# B&R Automation Studio project MotionProyect (part 2)

#### basicCyclic.st - cyclic code
```iecst
(********************************************************************
 * COPYRIGHT -- Bernecker + Rainer
 ********************************************************************
 * PROGRAM: Basic
 * File: basicCyclic.st
 * Author: Bernecker + Rainer
 * Created: December 01, 2009
 ********************************************************************
 * Implementation of Program Basic
 ********************************************************************)
PROGRAM _CYCLIC

(***************************************************************
        Control Sequence
***************************************************************)
	Axis2Cmd;
	Axis2Param;
	Axis2CyclicReadAction;

(* status information is read before the step sequencer to attain a shorter reaction time *)
(************************ MC_READSTATUS *************************)
MC_ReadStatus_0.Enable := NOT(MC_ReadStatus_0.Error);
MC_ReadStatus_0.Axis := Axis1Obj;
MC_ReadStatus_0();
BasicControl.AxisState.Disabled             := MC_ReadStatus_0.Disabled;
BasicControl.AxisState.StandStill           := MC_ReadStatus_0.StandStill;
BasicControl.AxisState.Stopping             := MC_ReadStatus_0.Stopping;
BasicControl.AxisState.Homing               := MC_ReadStatus_0.Homing;
BasicControl.AxisState.DiscreteMotion       := MC_ReadStatus_0.DiscreteMotion;
BasicControl.AxisState.ContinuousMotion     := MC_ReadStatus_0.ContinuousMotion;
BasicControl.AxisState.SynchronizedMotion   := MC_ReadStatus_0.SynchronizedMotion;
BasicControl.AxisState.ErrorStop            := MC_ReadStatus_0.Errorstop;

(********************MC_BR_READDRIVESTATUS***********************)
MC_BR_ReadDriveStatus_0.Enable := NOT(MC_BR_ReadDriveStatus_0.Error);
MC_BR_ReadDriveStatus_0.Axis := Axis1Obj;
MC_BR_ReadDriveStatus_0.AdrDriveStatus := ADR(BasicControl.Status.DriveStatus);
MC_BR_ReadDriveStatus_0();

(******************** MC_READACTUALPOSITION *********************)
MC_ReadActualPosition_0.Enable := (NOT(MC_ReadActualPosition_0.Error));
MC_ReadActualPosition_0.Axis := Axis1Obj;
MC_ReadActualPosition_0();
IF(MC_ReadActualPosition_0.Valid = TRUE)THEN
    BasicControl.Status.ActPosition := MC_ReadActualPosition_0.Position;
END_IF

(******************** MC_READACTUALVELOCITY *********************)
MC_ReadActualVelocity_0.Enable := (NOT(MC_ReadActualVelocity_0.Error));
MC_ReadActualVelocity_0.Axis := Axis1Obj;
MC_ReadActualVelocity_0();
IF(MC_ReadActualVelocity_0.Valid = TRUE)THEN
    BasicControl.Status.ActVelocity := MC_ReadActualVelocity_0.Velocity;
END_IF

(************************ MC_READAXISERROR **********************)
MC_ReadAxisError_0.Enable := NOT(MC_ReadAxisError_0.Error);
MC_ReadAxisError_0.Axis := Axis1Obj;
MC_ReadAxisError_0.DataAddress := ADR(BasicControl.Status.ErrorText);
MC_ReadAxisError_0.DataLength := SIZEOF(BasicControl.Status.ErrorText);
MC_ReadAxisError_0.DataObjectName := 'acp10etxen';
MC_ReadAxisError_0();

(**************** CHECK FOR GENERAL AXIS ERROR ******************)
    IF ((MC_ReadAxisError_0.AxisErrorID <> 0) AND (MC_ReadAxisError_0.Valid = TRUE)) THEN
        AxisStep := STATE_ERROR_AXIS;
(***************** CHECK IF POWER SHOULD BE OFF *******************)
    ELSIF ((BasicControl.Command.Power = FALSE) AND (MC_ReadAxisError_0.Valid = TRUE)) THEN
        IF ((MC_ReadStatus_0.Errorstop = TRUE) AND (MC_ReadStatus_0.Valid = TRUE)) THEN
            AxisStep := STATE_ERROR_RESET;
        ELSE
            AxisStep := STATE_WAIT;
        END_IF
    END_IF

(* central monitoring OF stop command attains a shorter reaction TIME in CASE OF emergency stop *)
(******************CHECK FOR STOP COMMAND************************)
    IF (BasicControl.Command.Stop = TRUE) THEN
        IF ((AxisStep >= STATE_HOME) AND (AxisStep <= STATE_ERROR)) THEN
            (* reset all FB execute inputs we use *)
            MC_Home_0.Execute := 0;
            MC_Stop_0.Execute := 0;
            MC_MoveAbsolute_0.Execute := 0;
            MC_MoveAdditive_0.Execute := 0;
            MC_MoveVelocity_0.Execute := 0;
            MC_ReadAxisError_0.Acknowledge := 0;
            MC_Reset_0.Execute := 0;
            MC_Halt_0.Execute := 0;

            (* reset user commands *)
            BasicControl.Command.Halt := 0;
            BasicControl.Command.Home := 0;
            BasicControl.Command.MoveJogPos := 0;
            BasicControl.Command.MoveJogNeg := 0;
            BasicControl.Command.MoveVelocity := 0;
            BasicControl.Command.MoveAbsolute := 0;
            BasicControl.Command.MoveAdditive := 0;
            AxisStep := STATE_STOP;
        END_IF
    END_IF

CASE AxisStep OF

(******************** WAIT *************************)
    STATE_WAIT:  (* STATE: Wait *)
        IF (BasicControl.Command.Power = TRUE) THEN
            AxisStep := STATE_POWER_ON;
        ELSE
            MC_Power_0.Enable := FALSE;
        END_IF

        (* reset all FB execute inputs we use *)
        MC_Home_0.Execute := FALSE;
        MC_Stop_0.Execute := FALSE;
        MC_MoveAbsolute_0.Execute := FALSE;
        MC_MoveAdditive_0.Execute := FALSE;
        MC_MoveVelocity_0.Execute := FALSE;
        MC_Halt_0.Execute := FALSE;
        MC_ReadAxisError_0.Acknowledge := FALSE;
        MC_Reset_0.Execute := FALSE;

        (* reset user commands *)
        BasicControl.Command.Stop := FALSE;
        BasicControl.Command.Halt := FALSE;
        BasicControl.Command.Home := FALSE;
        BasicControl.Command.MoveJogPos := FALSE;
        BasicControl.Command.MoveJogNeg := FALSE;
        BasicControl.Command.MoveVelocity := FALSE;
        BasicControl.Command.MoveAbsolute := FALSE;
        BasicControl.Command.MoveAdditive := FALSE;

        BasicControl.Status.ErrorID := 0;

(******************** POWER ON **********************)
    STATE_POWER_ON:  (* STATE: Power on *)
        MC_Power_0.Enable := TRUE;
        IF (MC_Power_0.Status = TRUE) THEN
            AxisStep := STATE_READY;
        END_IF
        (* if a power error occured go to error state *)
        IF (MC_Power_0.Error = TRUE) THEN
            BasicControl.Status.ErrorID := MC_Power_0.ErrorID;
            AxisStep := STATE_ERROR;
        END_IF

(******************** READY **********************)
    STATE_READY:  (* STATE: Waiting for commands *)
        IF (BasicControl.Command.Home = TRUE)THEN
            BasicControl.Command.Home := FALSE;
            AxisStep := STATE_HOME;

        ELSIF (BasicControl.Command.Stop = TRUE) THEN
            AxisStep := STATE_STOP;

        ELSIF (BasicControl.Command.MoveJogPos = TRUE) THEN
            AxisStep := STATE_JOG_POSITIVE;

        ELSIF (BasicControl.Command.MoveJogNeg = TRUE) THEN
            AxisStep := STATE_JOG_NEGATIVE;

        ELSIF (BasicControl.Command.MoveAbsolute = TRUE) THEN
            BasicControl.Command.MoveAbsolute := FALSE;
            AxisStep := STATE_MOVE_ABSOLUTE;

        ELSIF (BasicControl.Command.MoveAdditive = TRUE) THEN
            BasicControl.Command.MoveAdditive := FALSE;
            AxisStep := STATE_MOVE_ADDITIVE;

        ELSIF (BasicControl.Command.MoveVelocity = TRUE) THEN
            BasicControl.Command.MoveVelocity := FALSE;
            AxisStep := STATE_MOVE_VELOCITY;

        ELSIF (BasicControl.Command.Halt = TRUE) THEN
            BasicControl.Command.Halt := FALSE;
            AxisStep := STATE_HALT;
        END_IF

(******************** HOME **********************)
    STATE_HOME:  (* STATE: start homing process *)
        MC_Home_0.Position := BasicControl.Parameter.HomePosition;
        MC_Home_0.HomingMode := BasicControl.Parameter.HomeMode;
        MC_Home_0.Execute := TRUE;
        IF (MC_Home_0.Done = TRUE) THEN
            MC_Home_0.Execute := FALSE;
            AxisStep := STATE_READY;
        END_IF
        (* if a homing error occured go to error state *)
        IF (MC_Home_0.Error = TRUE) THEN
            MC_Home_0.Execute := FALSE;
            BasicControl.Status.ErrorID := MC_Home_0.ErrorID;
            AxisStep := STATE_ERROR;
        END_IF

(***********************HALT_MOVEMENT***************************)
    STATE_HALT:   (* STATE: Halt movement *)
        MC_Halt_0.Deceleration := BasicControl.Parameter.Deceleration;
        MC_Halt_0.Execute := TRUE;
        IF (MC_Halt_0.Done = TRUE) THEN
            MC_Halt_0.Execute := FALSE;
            AxisStep := STATE_READY;
        END_IF
        (* check if error occured *)
        IF (MC_Halt_0.Error = TRUE) THEN
            BasicControl.Status.ErrorID := MC_Halt_0.ErrorID;
            MC_Halt_0.Execute := FALSE;
            AxisStep := STATE_ERROR;
        END_IF

(*********************** STOP MOVEMENT *************************)
    STATE_STOP:  (* STATE: Stop movement *)
        MC_Stop_0.Deceleration := BasicControl.Parameter.Deceleration;
        MC_Stop_0.Execute := TRUE;
        (* if axis is stopped go to ready state *)
        IF ((MC_Stop_0.Done = TRUE) AND (BasicControl.Command.Stop = FALSE)) THEN
            MC_Stop_0.Execute := FALSE;
            AxisStep := STATE_READY;
        END_IF
        (* check if error occured *)
        IF (MC_Stop_0.Error = TRUE) THEN
            BasicControl.Status.ErrorID := MC_Stop_0.ErrorID;
            MC_Stop_0.Execute := FALSE;
            AxisStep := STATE_ERROR;
        END_IF

(******************** START JOG MOVEMENT POSITVE **********************)
     STATE_JOG_POSITIVE:  (* STATE: Start jog movement in positive direction *)
        MC_MoveVelocity_0.Velocity      := BasicControl.Parameter.JogVelocity;
        MC_MoveVelocity_0.Acceleration  := BasicControl.Parameter.Acceleration;
        MC_MoveVelocity_0.Deceleration  := BasicControl.Parameter.Deceleration;
        MC_MoveVelocity_0.Direction     := mcPOSITIVE_DIR;
        MC_MoveVelocity_0.Execute := TRUE;
        IF (BasicControl.Command.MoveJogPos = FALSE) THEN
            MC_MoveVelocity_0.Execute := FALSE;
            AxisStep := STATE_HALT;
        END_IF
        (* check if error occured *)
        IF (MC_MoveVelocity_0.Error = TRUE) THEN
            BasicControl.Status.ErrorID := MC_MoveVelocity_0.ErrorID;
            MC_MoveVelocity_0.Execute := FALSE;
            AxisStep := STATE_ERROR;
        END_IF

(******************** START JOG MOVEMENT NEGATIVE **********************)
    STATE_JOG_NEGATIVE:  (* STATE: Start jog movement in negative direction *)
        MC_MoveVelocity_0.Velocity      := BasicControl.Parameter.JogVelocity;
        MC_MoveVelocity_0.Acceleration  := BasicControl.Parameter.Acceleration;
        MC_MoveVelocity_0.Deceleration  := BasicControl.Parameter.Deceleration;
        MC_MoveVelocity_0.Direction	    := mcNEGATIVE_DIR;
        MC_MoveVelocity_0.Execute := TRUE;
        IF (BasicControl.Command.MoveJogNeg = FALSE) THEN
            MC_MoveVelocity_0.Execute := FALSE;
            AxisStep := STATE_HALT;
        END_IF
        (* check if error occured *)
        IF (MC_MoveVelocity_0.Error = TRUE) THEN
            BasicControl.Status.ErrorID := MC_MoveVelocity_0.ErrorID;
            MC_MoveVelocity_0.Execute := FALSE;
            AxisStep := STATE_ERROR;
        END_IF

(******************** START ABSOLUTE MOVEMENT **********************)
     STATE_MOVE_ABSOLUTE:  (* STATE: Start absolute movement *)
        MC_MoveAbsolute_0.Position      := BasicControl.Parameter.Position;
        MC_MoveAbsolute_0.Velocity      := BasicControl.Parameter.Velocity;
        MC_MoveAbsolute_0.Acceleration  := BasicControl.Parameter.Acceleration;
        MC_MoveAbsolute_0.Deceleration  := BasicControl.Parameter.Deceleration;
        MC_MoveAbsolute_0.Direction     := BasicControl.Parameter.Direction;
        MC_MoveAbsolute_0.Execute := TRUE;
        (* check if commanded position is reached *)
        IF (BasicControl.Command.Halt) THEN
            BasicControl.Command.Halt := FALSE;
            MC_MoveAbsolute_0.Execute := FALSE;
            AxisStep := STATE_HALT;
        ELSIF (MC_MoveAbsolute_0.Done = TRUE) THEN
            MC_MoveAbsolute_0.Execute := FALSE;
            AxisStep := STATE_READY;
        END_IF
        (* check if error occured *)
        IF (MC_MoveAbsolute_0.Error = TRUE) THEN
            BasicControl.Status.ErrorID := MC_MoveAbsolute_0.ErrorID;
            MC_MoveAbsolute_0.Execute := FALSE;
            AxisStep := STATE_ERROR;
        END_IF

(******************** START ADDITIVE MOVEMENT **********************)
    STATE_MOVE_ADDITIVE:  (* STATE: Start additive movement *)
        MC_MoveAdditive_0.Distance      := BasicControl.Parameter.Distance;
        MC_MoveAdditive_0.Velocity      := BasicControl.Parameter.Velocity;
        MC_MoveAdditive_0.Acceleration  := BasicControl.Parameter.Acceleration;
        MC_MoveAdditive_0.Deceleration  := BasicControl.Parameter.Deceleration;
        MC_MoveAdditive_0.Execute := TRUE;
        (* check if commanded distance is reached *)
        IF (BasicControl.Command.Halt) THEN
            BasicControl.Command.Halt := FALSE;
            MC_MoveAdditive_0.Execute := FALSE;
            AxisStep := STATE_HALT;
        ELSIF (MC_MoveAdditive_0.Done = TRUE) THEN
            MC_MoveAdditive_0.Execute := FALSE;
            AxisStep := STATE_READY;
        END_IF
        (* check if error occured *)
        IF (MC_MoveAdditive_0.Error = TRUE) THEN
            BasicControl.Status.ErrorID := MC_MoveAdditive_0.ErrorID;
            MC_MoveAdditive_0.Execute := FALSE;
            AxisStep := STATE_ERROR;
        END_IF

(******************** START VELOCITY MOVEMENT **********************)
    STATE_MOVE_VELOCITY:  (* STATE: Start velocity movement *)
        MC_MoveVelocity_0.Velocity      := BasicControl.Parameter.Velocity;
        MC_MoveVelocity_0.Acceleration  := BasicControl.Parameter.Acceleration;
        MC_MoveVelocity_0.Deceleration  := BasicControl.Parameter.Deceleration;
        MC_MoveVelocity_0.Direction     := BasicControl.Parameter.Direction;
        MC_MoveVelocity_0.Execute := TRUE;
        (* check if commanded velocity is reached *)
        IF (BasicControl.Command.Halt) THEN
            BasicControl.Command.Halt := FALSE;
            MC_MoveVelocity_0.Execute := FALSE;
            AxisStep := STATE_HALT;
        ELSIF (MC_MoveVelocity_0.InVelocity = TRUE) THEN
            MC_MoveVelocity_0.Execute := FALSE;
            AxisStep := STATE_READY;
        END_IF
        (* check if error occured *)
        IF (MC_MoveVelocity_0.Error = TRUE) THEN
            BasicControl.Status.ErrorID := MC_MoveVelocity_0.ErrorID;
            MC_MoveVelocity_0.Execute := FALSE;
            AxisStep := STATE_ERROR;
        END_IF

(******************** FB-ERROR OCCURED *************************)
    STATE_ERROR:  (* STATE: Error *)
        (* check if FB indicates an axis error *)
        IF (MC_ReadAxisError_0.AxisErrorCount<>0) THEN
            AxisStep := STATE_ERROR_AXIS;
        ELSE
            IF (BasicControl.Command.ErrorAcknowledge = TRUE) THEN
                BasicControl.Command.ErrorAcknowledge := FALSE;
                BasicControl.Status.ErrorID := 0;
                (* reset axis if it is in axis state ErrorStop *)
                IF ((MC_ReadStatus_0.Errorstop = TRUE) AND (MC_ReadStatus_0.Valid = TRUE)) THEN
                    AxisStep := STATE_ERROR_RESET;
                ELSE
                    AxisStep := STATE_WAIT;
                END_IF
            END_IF
        END_IF

(******************** AXIS-ERROR OCCURED *************************)
    STATE_ERROR_AXIS:  (* STATE: Axis Error *)
        IF (MC_ReadAxisError_0.Valid = TRUE) THEN
            IF (MC_ReadAxisError_0.AxisErrorID <> 0) THEN
                BasicControl.Status.ErrorID := MC_ReadAxisError_0.AxisErrorID;
            END_IF
            MC_ReadAxisError_0.Acknowledge := FALSE;
            IF (BasicControl.Command.ErrorAcknowledge = TRUE) THEN
                BasicControl.Command.ErrorAcknowledge := FALSE;
                (* acknowledge axis error *)
                IF (MC_ReadAxisError_0.AxisErrorID <> 0) THEN
                    MC_ReadAxisError_0.Acknowledge := TRUE;
                END_IF
            END_IF
            IF (MC_ReadAxisError_0.AxisErrorCount = 0) THEN
                (* reset axis if it is in axis state ErrorStop *)
                BasicControl.Status.ErrorID := 0;
                IF ((MC_ReadStatus_0.Errorstop = TRUE) AND (MC_ReadStatus_0.Valid = TRUE)) THEN
                    AxisStep := STATE_ERROR_RESET;
                ELSE
                    AxisStep := STATE_WAIT;
                END_IF
            END_IF
        END_IF

(******************** RESET DONE *************************)
    STATE_ERROR_RESET:  (* STATE: Wait for reset done *)
        MC_Reset_0.Execute := TRUE;
        (* reset MC_Power.Enable if this FB is in Error*)
        IF (MC_Power_0.Error = TRUE) THEN
            MC_Power_0.Enable := FALSE;
        END_IF
        IF(MC_Reset_0.Done = TRUE)THEN
            MC_Reset_0.Execute := FALSE;
            AxisStep := STATE_WAIT;
        ELSIF(MC_Reset_0.Error = TRUE) THEN
            MC_Reset_0.Execute := FALSE;
            AxisStep := STATE_ERROR;
        END_IF
(******************** SEQUENCE END *************************)
END_CASE

	AutoSequence.status.actPositon[2]		:= BasicControl.Status.ActPosition;
	AutoSequence.status.homingDone[2]		:= MC_Home_0.Done;
	AutoSequence.status.MoveAdditiveDone[2]	:= MC_MoveAdditive_0.Done;
	AutoSequence.status.moveAbsoluteDone[2]	:= MC_MoveAbsolute_0.Done;

	//ERROR OCCURRED
	IF BasicControl.Status.ErrorID <> 0 THEN
		AutoSequence.status.errorActive[2]	:= TRUE;
	ELSE
		AutoSequence.status.errorActive[2]	:= FALSE;
	END_IF;
(***************************************************************
        Function Block Calls
***************************************************************)

(************************** MC_POWER ****************************)
MC_Power_0.Axis := Axis1Obj;  (* pointer to axis *)
MC_Power_0();

(************************** MC_HOME *****************************)
MC_Home_0.Axis := Axis1Obj;
MC_Home_0();

(********************** MC_MOVEABSOLUTE *************************)
MC_MoveAbsolute_0.Axis := Axis1Obj;
MC_MoveAbsolute_0();

(********************** MC_MOVEADDITIVE *************************)
MC_MoveAdditive_0.Axis := Axis1Obj;
MC_MoveAdditive_0();

(********************** MC_MOVEVELOCITY *************************)
MC_MoveVelocity_0.Axis := Axis1Obj;
MC_MoveVelocity_0();

(************************** MC_STOP *****************************)
MC_Stop_0.Axis := Axis1Obj;
MC_Stop_0();

(***************************MC_HALT******************************)
MC_Halt_0.Axis := Axis1Obj;
MC_Halt_0();

(************************** MC_RESET ****************************)
MC_Reset_0.Axis := Axis1Obj;
MC_Reset_0();

END_PROGRAM
```

#### basicInit.st - init code
```iecst
PROGRAM _INIT

(* get axis object *)
Axis1Obj := ADR(gAxis02);

AxisStep := STATE_WAIT; (* start step *)

BasicControl.Parameter.Velocity             := 1000;  (*velocity for movement*)
BasicControl.Parameter.Acceleration         := 5000;  (*acceleration for movement*)
BasicControl.Parameter.Deceleration         := 5000;  (*deceleration for movement*)
BasicControl.Parameter.JogVelocity          := 400;   (*velocity for jogging *)

//	MC_BR_CyclicRead_0.Axis			:= ADR(gAxis02);
//	MC_BR_CyclicRead_0.Enable		:= TRUE;
//	MC_BR_CyclicRead_0.ParID		:= 381; //Temperature sensor: Temperature
//	MC_BR_CyclicRead_0.DataAddress	:= ADR(Axis1SensorTemp);
//	MC_BR_CyclicRead_0.DataType		:= ncPAR_TYP_REAL;
//	MC_BR_CyclicRead_0.Mode			:= mcEVERY_RECORD;
//	MC_BR_CyclicRead_0();
//
//
//	MC_BR_CyclicRead_1.Axis			:= ADR(gAxis02);
//	MC_BR_CyclicRead_1.Enable		:= TRUE;
//	MC_BR_CyclicRead_1.ParID		:= 1637; //Temperature sensor: Temperature
//	MC_BR_CyclicRead_1.DataAddress	:= ADR(Axis1MotorTorque);
//	MC_BR_CyclicRead_1.DataType		:= ncPAR_TYP_UINT;
//	MC_BR_CyclicRead_1.Mode			:= mcEVERY_RECORD;
//	MC_BR_CyclicRead_1();
END_PROGRAM
```

#### basic.var - Local variables
```iecst
VAR
	BasicControl : basic_typ; (*control structure*)
	MC_Home_0 : MC_Home; (*Function Block*)
	MC_MoveAbsolute_0 : MC_MoveAbsolute; (*Function Block*)
	MC_MoveAdditive_0 : MC_MoveAdditive; (*Function Block*)
	MC_MoveVelocity_0 : MC_MoveVelocity; (*Function Block*)
	MC_Power_0 : MC_Power; (*Function Block*)
	MC_ReadActualPosition_0 : MC_ReadActualPosition; (*Function Block *)
	MC_ReadActualVelocity_0 : MC_ReadActualVelocity; (*Function Block*)
	MC_ReadAxisError_0 : MC_ReadAxisError; (*Function Block*)
	MC_ReadStatus_0 : MC_ReadStatus; (*Function Block*)
	MC_Reset_0 : MC_Reset; (*Function Block*)
	MC_Stop_0 : MC_Stop; (*Function Block*)
	MC_BR_ReadDriveStatus_0 : MC_BR_ReadDriveStatus; (*Function Block*)
	MC_Halt_0 : MC_Halt; (*Function Block*)
	Axis1Obj : UDINT; (*axis reference*)
	AxisStep : UINT; (*current step in the step sequence*)
END_VAR
VAR CONSTANT
	STATE_READY : USINT := 10; (*constant for a waiting step*)
	STATE_POWER_ON : USINT := 1; (*constant for the step in which the controller is switched on*)
	STATE_MOVE_VELOCITY : USINT := 16; (*constant for the step in which a movement with defiened velocity is started*)
	STATE_MOVE_ABSOLUTE : USINT := 14; (*constant for the step in which a movement to defiened position is started*)
	STATE_WAIT : USINT := 0; (*constant for a waiting step*)
	STATE_STOP : USINT := 11; (*constant for the step in which movements are stopped*)
	STATE_MOVE_ADDITIVE : USINT := 15; (*constant for the step in which a movement with defiened distance is started*)
	STATE_HOME : USINT := 2; (*constant for the step in which the axis is homed*)
	STATE_ERROR_RESET : USINT := 102; (*constant for the step in which the errors are reset*)
	STATE_ERROR_AXIS : USINT := 100; (*constant for the axis error step*)
	STATE_ERROR : USINT := 101; (*constant for the error step*)
	STATE_JOG_POSITIVE : USINT := 12; (*constant for the step in which a positive jogging movement is executed*)
	STATE_JOG_NEGATIVE : USINT := 13; (*constant for the step in which a negative jogging movement is executed*)
	STATE_HALT : USINT := 17; (*constant for the step in which movements are stopped*)
END_VAR
VAR
	MC_BR_CyclicRead_0 : MC_BR_CyclicRead;
	MC_BR_CyclicRead_1 : MC_BR_CyclicRead;
	MC_BR_CyclicRead_2 : MC_BR_CyclicRead;
	Axis2SensorTemp : REAL;
	Axis2MotorTorque : REAL;
	Axis2EncoderPosition : DINT;
END_VAR
```

#### BasicAxis2Action.st
```iecst
ACTION Axis2CyclicReadAction:
	MC_BR_CyclicRead_0.Axis			:= ADR(gAxis02);
	MC_BR_CyclicRead_0.Enable		:= TRUE;
	MC_BR_CyclicRead_0.ParID		:= ACP10PAR_TEMP_MOTOR; //Temperature sensor: Temperature
	MC_BR_CyclicRead_0.DataAddress	:= ADR(Axis2SensorTemp);
	MC_BR_CyclicRead_0.DataType		:= ncPAR_TYP_REAL;
	MC_BR_CyclicRead_0.Mode			:= mcEVERY_RECORD;
	MC_BR_CyclicRead_0();

	MC_BR_CyclicRead_1.Axis			:= ADR(gAxis02);
	MC_BR_CyclicRead_1.Enable		:= TRUE;
	MC_BR_CyclicRead_1.ParID		:= ACP10PAR_TORQUE_ACT;
	MC_BR_CyclicRead_1.DataAddress	:= ADR(Axis2MotorTorque);
	MC_BR_CyclicRead_1.DataType		:= ncPAR_TYP_REAL;
	MC_BR_CyclicRead_1.Mode			:= mcEVERY_RECORD;
	MC_BR_CyclicRead_1();

	MC_BR_CyclicRead_2.Axis			:= ADR(gAxis02);
	MC_BR_CyclicRead_2.Enable		:= TRUE;
	MC_BR_CyclicRead_2.ParID		:= ACP10PAR_PCTRL_S_ACT;
	MC_BR_CyclicRead_2.DataAddress	:= ADR(Axis2EncoderPosition);
	MC_BR_CyclicRead_2.DataType		:= ncPAR_TYP_DINT;
	MC_BR_CyclicRead_2.Mode			:= mcEVERY_RECORD;
	MC_BR_CyclicRead_2();

END_ACTION

ACTION Axis2Param :
	BasicControl.Parameter.Acceleration	:= AutoSequence.par.acceleration;
	BasicControl.Parameter.Deceleration	:= AutoSequence.par.deceleration;
	BasicControl.Parameter.Direction	:= AutoSequence.par.direction[2];
	BasicControl.Parameter.Velocity		:= AutoSequence.par.speedMovement;
	BasicControl.Parameter.Distance		:= AutoSequence.par.distance[2];
	BasicControl.Parameter.HomePosition	:= AutoSequence.par.homePosition[2];
	BasicControl.Parameter.Position		:= AutoSequence.par.position[2];
END_ACTION

ACTION Axis2Cmd :
	BasicControl.Command.Power				:= AutoSequence.cmd.powerMotor;
	BasicControl.Command.Home				:= AutoSequence.cmd.home;
	BasicControl.Command.MoveAbsolute		:= AutoSequence.cmd.moveAbsolute[2];
	BasicControl.Command.MoveAdditive		:= AutoSequence.cmd.moveRelative[2];
	BasicControl.Command.Stop				:= AutoSequence.cmd.stopMotor;
	BasicControl.Command.ErrorAcknowledge	:= AutoSequence.cmd.ErrorAcknowledge[2];
END_ACTION
```

- Visualisation Logical/VC4/Visu (not shown)

- Visualisation Logical/VC4/VisuCtrl (not shown)

### Program Logical/VC4/VisCtrl

#### Variables.var
```iecst
VAR
	ShapeColor : ARRAY[1..3] OF USINT;
	i : USINT;
END_VAR
```

#### Main.st
```iecst
PROGRAM _INIT
	(* Insert code here *)

END_PROGRAM

PROGRAM _CYCLIC
	//Shape Colors
	FOR i := 1 TO 3 DO
		IF AutoSequence.status.doErrorActive THEN
			ShapeColor[i]	:= 253; //naranja
		ELSE
			ShapeColor[i]; //Negro
		END_IF	;

	END_FOR;

	IF AutoSequence.status.doPowerMotorsOff THEN
		ShapeColor[1]	:= 15; //Blanco
	ELSIF AutoSequence.status.doPowerMotorsON THEN
		ShapeColor[1]	:= 10; //Verde
	ELSE
		ShapeColor[1]	:= 0;
	END_IF;

	IF AutoSequence.status.doStartCycleInactive THEN
		ShapeColor[2]	:= 15; //Blanco
	ELSIF AutoSequence.status.doStartCycleActive THEN
		ShapeColor[2]	:= 10; //Verde
	ELSE
		ShapeColor[2]	:= 0;
	END_IF;

	IF NOT(AutoSequence.cmd.AutoSequenceDisabled)  THEN
		IF (AutoSequence.status.doStopCycleActive) THEN
			ShapeColor[3]	:= 45;
		ELSIF NOT (AutoSequence.status.doStopCycleActive)  THEN
			ShapeColor[3]	:= 15;
		ELSE
			ShapeColor[3];
		END_IF;
	ELSIF (AutoSequence.cmd.AutoSequenceDisabled)  THEN
		IF 	AutoSequence.status.doManualMode THEN
				ShapeColor[3]	:=  206; //Azul
			ELSE
				ShapeColor[3]	:= 15; //Negro
			END_IF;
	END_IF;

END_PROGRAM

PROGRAM _EXIT
	(* Insert code here *)

END_PROGRAM
```

Listed in the project but not available here: Logical/Source/AxisCtrl/Types.typ, Logical/Sources/MotionControl/Types.typ, Logical/Sources/MotionControl/BasicAxis1/basic.typ, Logical/Sources/MotionControl/BasicAxis2/basic.typ
